// TIA Portal V17 export
// export: Created 2025-03-07T09:24:38.7273089Z, ExportSetting WithDefaults, DisplayName Totally Integrated Automation Portal, DisplayVersion V17 Update 8, DisplayName TIA Portal Openness, DisplayVersion V17 Update 8, DisplayName TIA Portal Version Control Interface, DisplayVersion V17, DisplayName SINAMICS Startdrive Advanced, DisplayVersion V17 SP2, DisplayName SINAMICS Startdrive G110M, G120, G120C, G120D, G120P, G115D, DisplayVersion V17 SP2, DisplayName SINAMICS Startdrive G130, G150, S120, S150, SINAMICS MV, S210, DisplayVersion V17 SP2, DisplayName STEP 7 Professional, DisplayVersion V17 Update 8, DisplayName SINUMERIK ONE STEP 7 Toolbox, DisplayVersion V17 Update 12, DisplayName SINUMERIK 840D sl STEP 7 Toolbox, DisplayVersion V17 Update 12, DisplayName STEP 7 Safety, DisplayVersion V17 Update 6, DisplayName WinCC Advanced, DisplayVersion V17 Update 8
TYPE "UNIT ALARM"
// stored: IsFailsafeCompliant false
   STRUCT
      IS_ALARMS : Bool;   // IMMEDIATE STOP ALARMS
      IS_SEOC_ALARMS : Bool;   // IMMEDIATE STOP & STOP END OF CYCLE ALARMS / IMMEDIATE STOP AND STOP END OF CYCLE ALARMS
      RHP_ALARMS : Bool;   // RETURN HOME POSITION ALARMS
      RHP_SEOC_ALARMS : Bool;   // RETURN HOME POSITION & STOP END OF CYCLE ALARMS / RETURN HOME POSITION AND STOP END OF CYCLE ALARMS
      SEOC_ALARMS : Bool;   // STOP END OF CYCLE ALARMS
      IS_WARNING : Bool;   // IMMEDIATE STOP WARNING / IMMEDIATE STOP WARNINGS
      RHP_WARNING : Bool;   // RETURN HOME POSITION WARNING / RETURN HOME POSITION WARNINGS
      SEOC_WARNING : Bool;   // STOP END OF CYCLE WARNING / STOP END OF CYCLE WARNINGS
      WARNING : Bool;   // WARNING / WARNINGS
      HELP : Bool;   // HELP
      ALARM : Bool;   // ALARM
      WARNING_STOP : Bool;   // WARNING STOP
      RESET_ALL_SEQUENCES : Bool;   // RESET ALL SEQUENCES
      RESET_LOCAL_SEQUENCES : Bool;   // RESET LOCAL SEQUENCES
      MASK_IS : Bool;   // MASK IMMEDIATE STOP
      MASK_IS_SEOC : Bool;   // MASK IMMEDIATE STOP & STOP END OF CYCLE / MASK IMMEDIATE STOP AND STOP END OF CYCLE
      MASK_RHP : Bool;   // MASK RETURN HOME POSITION
      MASK_RHP_SEOC : Bool;   // MASK RETURN HOME POSITION & STOP END OF CYCLE / MASK RETURN HOME POSITION AND STOP END OF CYCLE
      MASK_SEOC : Bool;   // MASK STOP END OF CYCLE
      MASK_IS_WARNING : Bool;   // MASK IMMEDIATE STOP WARNING
      MASK_RHP_WARNING : Bool;   // MASK RETURN HOME POSITIONS WARNING
      MASK_SEOC_WARNING : Bool;   // MASK STOP END OF CYCLE WARNING
      MASK_WARNING : Bool;   // MASK WARNING
      MASK_HELP : Bool;   // MASK HELP
      AUX_IS : Bool;   // AUXILIARY IMMEDIATE STOP ALARMS
      AUX_IS_SEOC : Bool;   // AUXILIARY IMMEDIATE STOP & STOP END OF CYCLE ALARMS / AUXILIARY IMMEDIATE STOP AND STOP END OF CYCLE ALARMS
      AUX_RHP : Bool;   // AUXILIARY RETURN HOME POSITION ALARMS
      AUX_RHP_SEOC : Bool;   // AUXILIARY RETURN HOME POSITION & STOP END OF CYCLE ALARMS / AUXILIARY RETURN HOME POSITION AND STOP END OF CYCLE ALARMS
      AUX_SEOC : Bool;   // AUXILIARY STOP END OF CYCLE ALARMS
      AUX_IS_WARNING : Bool;   // AUXILIARY IMMEDIATE STOP WARNING / AUXILIARY IMMEDIATE STOP WARNINGS
      AUX_RHP_WARNING : Bool;   // AUXILIARY RETURN HOME POSITION WARNING / AUXILIARY RETURN HOME POSITION WARNINGS
      AUX_SEOC_WARNING : Bool;   // AUXILIARY STOP END OF CYCLE WARNING / AUXILIARY STOP END OF CYCLE WARNINGS
      AUX_WARNING : Bool;   // AUXILIARY WARNING / AUXILIARY WARNINGS
      AUX_HELP : Bool;   // AUXILIARY HELP
   END_STRUCT;
END_TYPE
